//Status information specific to the cabinet PNOZ --> IPC, can be customized depending on cabinet
TYPE ST_MCC_CustomStatusIn :
STRUCT
    bit16_EStopExperimentOK: BIT; //The Expirement caves, bitEStopOK (MCC5)
    bit17_EStopOpticalOK: BIT; //The Optical caves, bitEStopOK (MCC3)
    bit18_EStopExternalOK: BIT; //The Selene Guides, bitEStopOK (MCC4) = bitEStopOK (MCC3) AND bitEStopOK (MCC5)
    bit19_Reserved: BIT;
    bit20_Reserved: BIT;
    bit21_Reserved: BIT;
    bit22_Reserved: BIT;
    bit23_Reserved: BIT;
    bit24_Reserved: BIT;
    bit25_Reserved: BIT;
    bit26_Reserved: BIT;
    bit27_Reserved: BIT;
    bit28_Reserved: BIT;
    bit29_Reserved: BIT;
    bit30_Reserved: BIT;
    bit31_Reserved: BIT;
END_STRUCT
END_TYPE

(* stored: Version 1.1.0.1
   DUT ST_MCC_CustomStatusIn: Id {3047c094-43cd-0281-2261-d5308c49a667} *)
